//==================================================================================================
//							Beckhoff Automation Poland
//									23.05.2017
//	Program obslugujacy proste alarmy historyczne.
//	W opcjach wizualizacji trzeba wybrac use uniceode strings i use current visu variable
// 	v1.0	|| TC v 3.1.4020.32		|| - pierwsza wersja
//==================================================================================================
PROGRAM P_EventsHS
VAR
	fbLocalSystemTime						: FB_LocalSystemTime;
	bEventTableSizeError					: BOOL;					// Niewlasciwy rozmiar tablicy zdarzen - sprawdz GVL_EHS.diNoOfEvents
	bEventDefinitionSizeError				: BOOL;					// Niewlasciwy rozmiar tablicy zdarzen - sprawdz GVL_EHS.diEventsDefinition
END_VAR

fbLocalSystemTime(bEnable:= TRUE, systemTime=> GVL_EHS.stActTime);
GVL_EHS.dtActTime 							:= SYSTEMTIME_TO_DT(GVL_EHS.stActTime);

P_EventsDefinitionHS ();

bEventDefinitionSizeError 					:= GVL_EHS.diEventsDefinition < 5 OR GVL_EHS.diEventsDefinition > 1000;
bEventTableSizeError 						:= GVL_EHS.diNoOfEvents < 5 OR GVL_EHS.diNoOfEvents > 1000;

IF NOT bEventDefinitionSizeError AND NOT bEventTableSizeError THEN
	IF fbLocalSystemTime.bValid THEN
		P_EventsHandlingHS();
	END_IF
	// Visu i filtry
	P_EventsVisuHS();	
END_IF

END_PROGRAM

(* stored: Version 1.1.0.1, ProductVersion 3.1.4022.12
   POU P_EventsHS: Id {3f9e00f1-4ce6-45f9-888c-1e9f9363e906}, SpecialFunc None *)
